// TIA Portal V19 export
TYPE "C501_VAR_IF_KLG_TYPIC"
   STRUCT
      STS_OPEN { ExternalAccessible := 'False'; ExternalVisible := 'False'; ExternalWritable := 'False'} : Bool;   // Motorgestuurde klep is open
      STS_TOE { ExternalAccessible := 'False'; ExternalVisible := 'False'; ExternalWritable := 'False'} : Bool;   // Motorgestuurde klep is toe
      STS_BEZ_OPEN { ExternalAccessible := 'False'; ExternalVisible := 'False'; ExternalWritable := 'False'} : Bool;   // Motorgestuurde klep is aan het openen (1 = Open)
      STS_BEZ_TOE { ExternalAccessible := 'False'; ExternalVisible := 'False'; ExternalWritable := 'False'} : Bool;   // Motorgestuurde klep is aan het sluiten (1 = Toe)
      BMO_HAND { ExternalAccessible := 'False'; ExternalVisible := 'False'; ExternalWritable := 'False'} : Bool;   // TRUE = in hand geschakeld FALSE = niet in hand
      EXT_HW { ExternalAccessible := 'False'; ExternalVisible := 'False'; ExternalWritable := 'False'} : Bool;   // Sturings hardware (PLC) in storing
      STO { ExternalAccessible := 'False'; ExternalVisible := 'False'; ExternalWritable := 'False'} : Struct   // Opsomming van alle storingen
         A001 : Bool;   // Beveiliging aangesproken
         AT01 : Bool;   // Terugmelding Open niet ontvangen
         AT02 : Bool;   // Terugmelding Dicht niet ontvangen
         AT03 : Bool;   // Terugmeldingen Open en Dicht tegelijkertijd
      END_STRUCT;
   END_STRUCT;
END_TYPE
